FUNCTION_BLOCK LampControl
VAR
	LampP1 AT%Q* : BOOL;
	_Control : ITF_Control;
END_VAR

PROPERTY Controller : ITF_Control
GET
Controller := _Control;
END_GET
SET
_Control := Controller;
END_SET
END_PROPERTY

METHOD Cycle : BOOL
VAR_INPUT
END_VAR
LampP1 := _Control.GetSwitchS10();
END_METHOD

END_FUNCTION_BLOCK

(* stored: Version 1.1.0.1, ProductVersion 3.1.4024.12
   POU LampControl: Id {df181268-03ef-4209-a1a2-ca82e29954b4}, SpecialFunc None
   Property Controller: Id {2f384581-c577-4ad4-a428-bd18dc912aa5}
   Get Get: Id {27b2ebad-7020-4771-9e8e-50cc5ac97c22}
   Set Set: Id {1139ded0-5cb7-4cda-aad5-86cdb67580cc}
   Method Cycle: Id {71ab4db3-ea61-4310-a4f0-cec5f96e91d9} *)
